Universal Robots PolyScope program: taskboard_belt_v5.urp

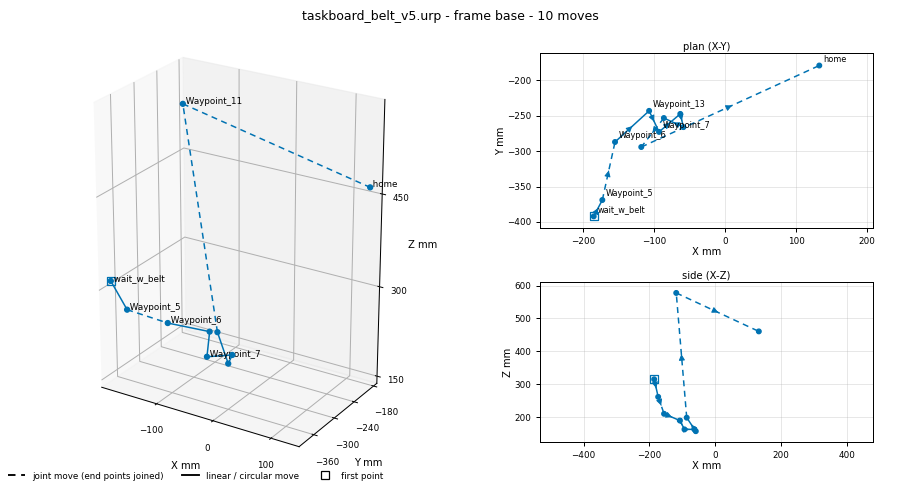
[picture p0: tool path of taskboard_belt_v5.urp in frame base, 10 of 10 moves have a stored position in this frame; points joined in program order, loops and branches not executed]
Program taskboard_belt_v5 (installation=default directory=/programs/wrs2020 createdIn=5.6.0.90886 lastSavedIn=5.9.1.1031110 robotSerialNumber=20205500180)
Calibrated DH parameters: a=[0, -0.425, -0.3922, 0, 0, 0]; d=[0.1625, 0, 0, 0.1333, 0.0997, 0.0996]; alpha=[1.570796, 0, 0, 1.570796, -1.570796, 0]; deltaTheta=[0, 0, 0, 0, 0, 0]
Robot Program (runOnlyOnce=true)
  SuppressedNode
    MoveJ speed 60 deg/s, acceleration 80 deg/s^2 (useActiveTCP=true) feature=Base
      currentpose := get_actual_joint_positions()
      Waypoint Waypoint (Variable): variable=currentpose
  MoveL speed 250 mm/s, acceleration 150 mm/s^2 (useActiveTCP=false) tcp=TCP; feature=Base
    SuppressedNode
      Waypoint above_tray: motionParameters(blendRadius=0.05); TCP in base x=-172.311 y=-492.624 z=406.821 mm, rx=2.0826 ry=-2.3042 rz=0.0252 rad; joints [55.84, -87.577, 100.035, -104.661, -89.581, -118.368] deg
    Waypoint wait_w_belt: TCP in base x=-185.572 y=-392.078 z=315.254 mm, rx=-1.4441 ry=1.9502 rz=-1.0486 rad; joints [37.028, -91.796, 114.934, -76.388, -46.414, -141.19] deg
  Popup Message (haltProgram=false message=start sequence together with b_bot (simultaneous start) inputType=Text)
  Wait Sleep waitTime=2.5
  MoveL speed 250 mm/s, acceleration 1200 mm/s^2 (useActiveTCP=false) tcp=TCP; feature=Base
    Waypoint Waypoint_5: TCP in base x=-173.43 y=-369.039 z=261.712 mm, rx=-1.282 ry=1.8047 rz=-1.1483 rad; joints [34.616, -88.409, 119.828, -68.558, -43.225, -150.47] deg
  MoveJ speed 60 deg/s, acceleration 80 deg/s^2 (useActiveTCP=false) tcp=TCP; feature=Base
    Waypoint Waypoint_6: TCP in base x=-155.523 y=-287.24 z=210.263 mm, rx=-1.031 ry=1.6203 rz=-1.5379 rad; joints [21.885, -87.537, 130.935, -50.465, -40.317, -177.586] deg
  MoveL speed 250 mm/s, acceleration 1200 mm/s^2 (useActiveTCP=false) tcp=TCP; feature=Base
    Waypoint Waypoint_13: TCP in base x=-107.458 y=-243.362 z=189.808 mm, rx=-0.909 ry=1.7261 rz=-1.6615 rad; joints [13.916, -96.788, 144.22, -53.106, -38.64, -178.723] deg
    Waypoint Waypoint_7: TCP in base x=-93.501 y=-273.032 z=162.831 mm, rx=-0.9044 ry=1.7298 rz=-1.6658 rad; joints [21.869, -90.172, 144.622, -61.38, -30.363, -177.16] deg
  Wait Sleep waitTime=1
  MoveL speed 250 mm/s, acceleration 1200 mm/s^2 (useActiveTCP=false) tcp=TCP; feature=Base
    Waypoint Waypoint_8: TCP in base x=-63.539 y=-247.671 z=163.129 mm, rx=-0.7441 ry=1.8696 rz=-1.7976 rad; joints [15.11, -101.236, 153.772, -59.958, -25.437, -176.345] deg
  MoveL speed 250 mm/s, acceleration 1200 mm/s^2 (useActiveTCP=false) tcp=TCP; feature=Base
    Waypoint Waypoint_9: TCP in base x=-59.125 y=-266.29 z=157.434 mm, rx=-0.7441 ry=1.8696 rz=-1.7976 rad; joints [21.298, -97.571, 152.76, -64.841, -19.306, -173.924] deg
  Wait Sleep waitTime=5
  URCap Gripper (Robotiq_Grippers, Robotiq Inc.) dataModel(position=80.3921568627451, force=0.0, speed=0.0, positionInDouble=80.3921568627451, forceInDouble=0.0, speedInDouble=0.0, slaveIds=[9], blocking=true)
  MoveL speed 250 mm/s, acceleration 1200 mm/s^2 (useActiveTCP=false) tcp=TCP; feature=Base
    Waypoint Waypoint_10: TCP in base x=-86.692 y=-253.478 z=198.507 mm, rx=-0.7729 ry=1.8477 rz=-1.7806 rad; joints [15.395, -103.398, 147.395, -51.019, -26.952, -177] deg; TCP offset x=0 y=0 z=0 mm, rx=0 ry=0 rz=0 rad
  MoveJ speed 120 deg/s, acceleration 100 deg/s^2 (useActiveTCP=false) tcp=TCP; feature=Base
    Waypoint Waypoint_11: TCP in base x=-118.553 y=-294.346 z=577.587 mm, rx=1.3176 ry=2.7241 rz=-0.2718 rad; joints [40.024, -118.444, 99.589, -78.038, -80.282, 2.128] deg
    Waypoint home: TCP in base x=132.399 y=-179.474 z=460.725 mm, rx=-0.0051 ry=-3.1414 rz=-0.0307 rad; joints [89.952, -120.316, 80.22, -48.701, -89.95, -0.003] deg; TCP offset x=0 y=0 z=220 mm, rx=0 ry=0 rz=0 rad
